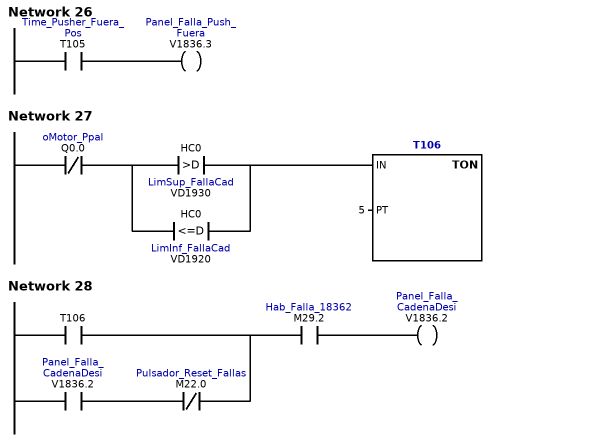
[picture p48: SBR20 networks 26-28]
Network 26
LD     Time_Pusher_Fuera_Pos:T105
=      Panel_Falla_Push_Fuera:V1836.3
Network 27
LDN    oMotor_Ppal:Q0.0
LDD>   HC0, LimSup_FallaCad:VD1930
OD<=   HC0, LimInf_FallaCad:VD1920
ALD
TON    T106, 5
Network 28
LD     T106
LD     Panel_Falla_CadenaDesi:V1836.2
AN     Pulsador_Reset_Fallas:M22.0
OLD
A      Hab_Falla_18362:M29.2
=      Panel_Falla_CadenaDesi:V1836.2
END_SUBROUTINE_BLOCK

SUBROUTINE_BLOCK Posiciones_Caja:SBR25
TITLE=
BEGIN
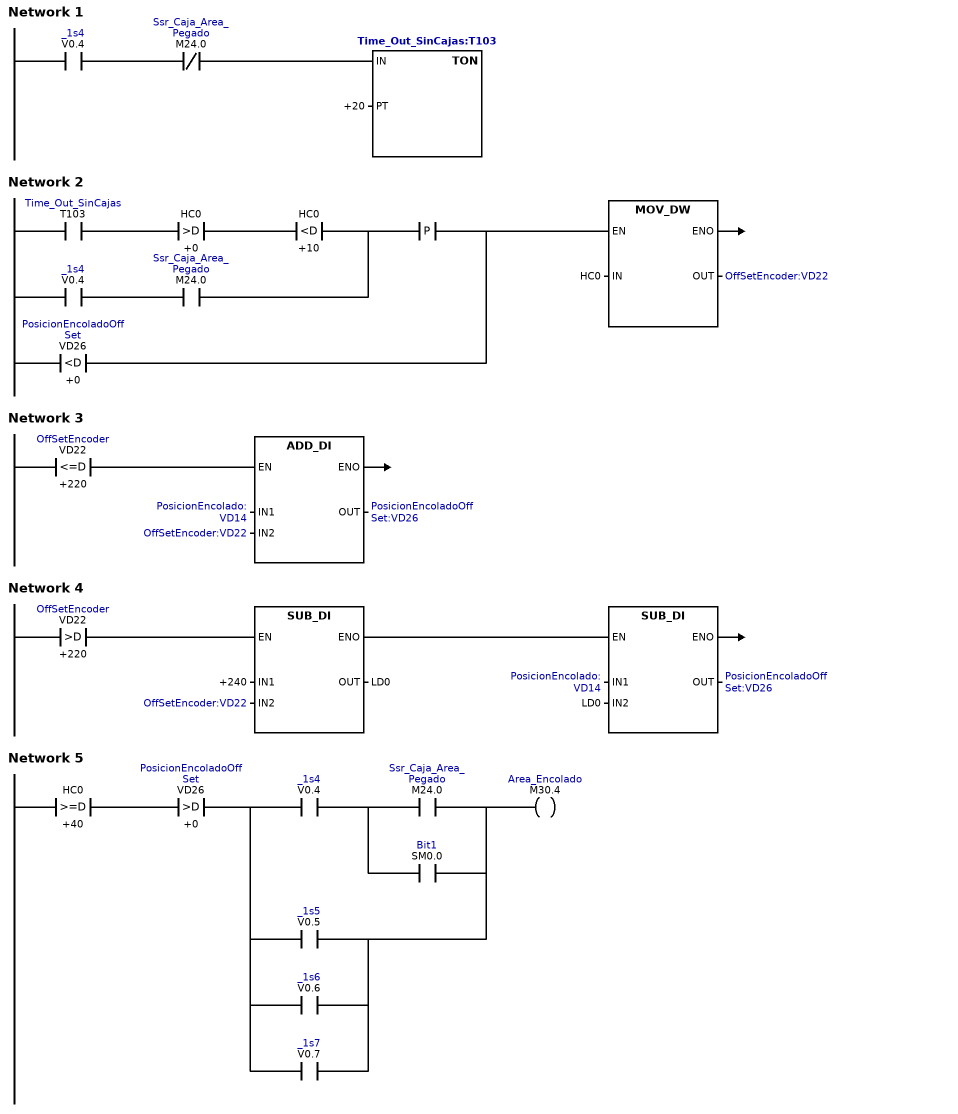
Network 1
LD     _1s4:V0.4
AN     Ssr_Caja_Area_Pegado:M24.0
TON    Time_Out_SinCajas:T103, +20
Network 2
LD     Time_Out_SinCajas:T103
AD>    HC0, +0
AD<    HC0, +10
LD     _1s4:V0.4
A      Ssr_Caja_Area_Pegado:M24.0
OLD
EU
OD<    PosicionEncoladoOffSet:VD26, +0
MOVD   HC0, OffSetEncoder:VD22
Network 3
LDD<=  OffSetEncoder:VD22, +220
MOVD   PosicionEncolado:VD14, PosicionEncoladoOffSet:VD26
+D     OffSetEncoder:VD22, PosicionEncoladoOffSet:VD26
Network 4
LDD>   OffSetEncoder:VD22, +220
MOVD   +240, LD0
AENO
-D     OffSetEncoder:VD22, LD0
AENO
MOVD   PosicionEncolado:VD14, PosicionEncoladoOffSet:VD26
-D     LD0, PosicionEncoladoOffSet:VD26
Network 5
LDD>=  HC0, +40
AD>    PosicionEncoladoOffSet:VD26, +0
LD     _1s4:V0.4
LD     Ssr_Caja_Area_Pegado:M24.0
O      Bit1:SM0.0
ALD
LD     _1s5:V0.5
O      _1s6:V0.6
O      _1s7:V0.7
OLD
ALD
=      Area_Encolado:M30.4
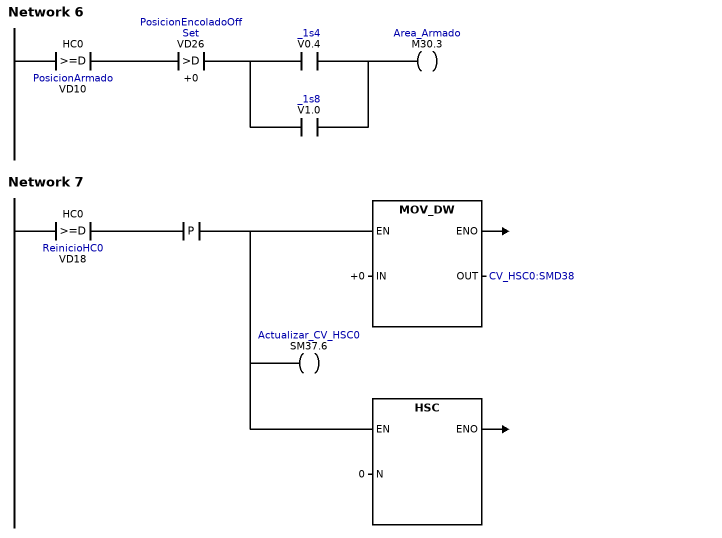
Network 6
LDD>=  HC0, PosicionArmado:VD10
AD>    PosicionEncoladoOffSet:VD26, +0
LD     _1s4:V0.4
O      _1s8:V1.0
ALD
=      Area_Armado:M30.3
Network 7
LDD>=  HC0, ReinicioHC0:VD18
EU
MOVD   +0, CV_HSC0:SMD38
=      Actualizar_CV_HSC0:SM37.6
HSC    0
END_SUBROUTINE_BLOCK

DATA_BLOCK_TAB USUARIO1
BEGIN
//COMENTARIOS DEL BLOQUE DE DATOS
//Pulse F1 para obtener Ayuda y un bloque de datos de ejemplo.
//****************************************************************
//****UTILIZO DE LAS WORDS DE 0 A 10 PARA LOS ESTADOS INTERNOS****
//****************************************************************
         _1sD1, 0            //Word de estados 1
         _2sw1, 0            //Word de estados 2
         _3sw1, 0            //Word de estados 3
         _4sw1, 0            //Word de estados 4
//****************************************************
//****UTILIZO DE LAS WORDS DE 10 A 100 PARA VARIOS****
//****************************************************
         PosicionArmado, 230 //Valor donde el encoder debe iniciar la secuencia de ARMADO
         PosicionEncolado, 5 //Valor donde el encoder debe iniciar la secuencia de PEGADO
         ReinicioHC0, 240    //Valor de reinicio del contador rapido HC0
         OffSetEncoder, 5    //Valor de Off set para cuentas encoder
         PosicionEncoladoOffSet, 0 //Valor para inicio Encolado con Off Set incluido
         WFallas, 0          //Word de FALLAS PARA PANEL!!!!
         Tiempo_Encolado_1, 9 //Tiempo x10ms de Encolado 1 en Uso
         Tiempo_Encolado_2, 7 //Tiempo x10ms de Encolado 2 en Uso
         Tiempo_NO_Encolar, 25 //Tiempo x10ms de NO ENCOLADO en Uso
//****************************************************
//Los tiempos en el panel tienen 2 decimales y el formato es entero
//por lo que el dato que envia el panel es multiplicado
//por 100 (ya que posee 2 decimales)
//y los timer tienen base de tiempo = 10ms por lo que no debo
//realizar ninguna cuenta auxiliar  
//En panel => 1,00 seg = 100 (dato al PLC)
//100 * 0.01 seg = 1 seg
//****************************************************
         Panel_Timer_Corte_Vacio, 5 //Tiempo de Corte de vacio desde panel
         Panel_Sel_Caja, 0   //Selección de Programa por Tipo de Caja
VW112    0                   //Libre
VW114    0                   //Libre
VW116    0                   //Libre
VW118    0                   //Libre
//**************************************************************************
// VD120  Utilizada para ver en el panel los valores actuales del encoder*** 
//**************************************************************************
VW124    0                   //Libre
VW126    0                   //Libre
VW128    0                   //Libre
//**********************************************************
//Estas words son para ajustar los tiempos
//mecanicos de la maquinas, aca figuran comentados
//pero en el programa se utilizan
//**********************************************************
         D_Pnel_T_Escuadre, 0 //Panel_TON_10 Timer Tiempo de Escuadre
         D_Pnel_T_RetardoPushe, 0 //Panel_TON_10 Timer Tiempo de Retardo de Pusher
         D_Pnel_T_Arranque_Bba, 10 //Panel_TON_100 Timer Tiempo Arranque Bomba Vacio
         D_Pnel_T_ArranqCyMPpal, 4 //Panel_TON_100 Timer Tiempo Arranque Cinta y Motor Ppal.
         D_Pnel_T_Falla_Pusher, 10 //Panel_TON_100 Timer Tiempo Falla Motor Pusher
         D_Pnel_T_FallaPistPush, 10 //Panel_TON_100 Timer Tiempo Falla Piston Pusher
//**********************************************************
// Valores de Encolado Ajustados desde Panel
// En este caso los datos llegan por 10ms como es la base del timer
//**********************************************************
         Panel_Tie_Enc_1_0, 9 //Tiempo x10ms de Encolado 1 Caja 15x1000
         Panel_Tie_Enc_2_0, 7 //Tiempo x10ms de Encolado 2 Caja 15x1000
         Panel_Tie_NoEnc_0, 25 //Tiempo x10ms de No Encolado Caja 15x1000
         Panel_Tie_Enc_1_1, 9 //Tiempo x10ms de Encolado 1 Caja 12x1500
         Panel_Tie_Enc_2_1, 7 //Tiempo x10ms de Encolado 2 Caja 12x1500
         Panel_Tie_NoEnc_1, 25 //Tiempo x10ms de No Encolado Caja 12x1500
         Panel_Tie_Enc_1_2, 9 //Tiempo x10ms de Encolado 1 Caja 12x1000
         Panel_Tie_Enc_2_2, 6 //Tiempo x10ms de Encolado 2 Caja 12x1000
         Panel_Tie_NoEnc_2, 18 //Tiempo x10ms de No Encolado Caja 12x1000
         Panel_Tie_Enc_1_3, 7 //Tiempo x10ms de Encolado 1 Caja 12x750
         Panel_Tie_Enc_2_3, 6 //Tiempo x10ms de Encolado 2 Caja 12x750
         Panel_Tie_NoEnc_3, 15 //Tiempo x10ms de No Encolado Caja 12x750
//*********************************************************************
// A PARTIR DE LA V1800 ARRANCO CON EL INTERCAMBIO DE DATOS CON EL PANEL 
// Ver simbolicos Standart Panel!!
//*********************************************************************
V1862    
V1862    
V1862    
V1862    
V1862    
V1862    
V1862    
V1862    
V1863    
V1863    
V1863    
V1863    
V1863    
V1863    
V1863    
V1863    
V1864    
V1864    
V1864    
V1864    
V1864    
V1864    
V1864    
V1864    
V1865    
V1865    
V1865    
V1865    
V1865    
V1865    
V1865    
V1865    
V1866    
V1866    
V1866    
V1866    
V1866    
V1866    
V1866    
V1866    
V1867    
V1867    
V1867    
V1867    
V1867    
V1867    
V1867    
V1867    
V1868    
V1868    
V1868    
V1868    
V1868    
V1868    
V1868    
V1868    
V1869    
V1869    
V1869    
V1869    
V1869    
V1869    
V1869    
V1869    
V1870    
V1870    
V1870    
V1870    
V1870    
V1870    
V1870    
V1870    
V1871    
V1871    
V1871    
V1871    
V1871    
V1871    
V1871    
V1871    
V1872    
V1872    
V1872    
V1872    
V1872    
V1872    
V1872    
V1872    
V1873    
V1873    
V1873    
V1873    
V1873    
V1873    
V1873    
V1873    
V1894    
V1894    
V1894    
V1894    
V1894    
V1894    
V1894    
V1894    
V1895    
V1895    
V1895    
V1895    
V1895    
V1895    
V1895    
V1895    
V1896    
V1896    
V1896    
V1896    
V1896    
V1896    
V1896    
V1896    
V1897    
V1897    
V1897    
V1897    
V1897    
V1897    
V1897    
V1897    
V1898    
V1898    
V1898    
V1898    
V1898    
V1898    
V1898    
V1898    
V1899    
V1899    
V1899    
V1899    
V1899    
V1899    
V1899    
V1899    
V1900    
V1900    
V1900    
V1900    
V1900    
V1900    
V1900    
V1900    
V1901    
V1901    
V1901    
V1901    
V1901    
V1901    
V1901    
V1901    
V1902    
V1902    
V1902    
V1902    
V1902    
V1902    
V1902    
V1902    
V1903    
V1903    
V1903    
V1903    
V1903    
V1903    
V1903    
V1903    
V1904    
V1904    
V1904    
V1904    
V1904    
V1904    
V1904    
V1904    
V1905    
V1905    
V1905    
V1905    
V1905    
V1905    
V1905    
V1905    
V1996    
V1996    
V1996    
V1996    
V1996    
V1996    
V1996    
V1996    
V1997    
V1997    
V1997    
V1997    
V1997    
V1997    
V1997    
V1997    
V1998    
V1998    
V1998    
V1998    
V1998    
V1998    
V1998    
V1998    
V1999    
V1999    
V1999    
V1999    
V1999    
V1999    
V1999    
V1999    
V2000    
V2000    
V2000    
V2000    
V2000    
V2000    
V2000    
V2000    
V2001    
V2001    
V2001    
V2001    
V2001    
V2001    
V2001    
V2001    
V2002    
V2002    
V2002    
V2002    
V2002    
V2002    
V2002    
V2002    
V2003    
V2003    
V2003    
V2003    
V2003    
V2003    
V2003    
V2003    
V2004    
V2004    
V2004    
V2004    
V2004    
V2004    
V2004    
V2004    
V2005    
V2005    
V2005    
V2005    
V2005    
V2005    
V2005    
V2005    
V2006    
V2006    
V2006    
V2006    
V2006    
V2006    
V2006    
V2006    
V2007    
V2007    
V2007    
V2007    
V2007    
V2007    
V2007    
V2007    
V2008    
V2008    
V2008    
V2008    
V2008    
V2008    
V2008    
V2008    
V2009    
V2009    
V2009    
V2009    
V2009    
V2009    
V2009    
V2009    
V2010    
V2010    
V2010    
V2010    
V2010    
V2010    
V2010    
V2010    
V2011    
V2011    
V2011    
V2011    
V2011    
V2011    
V2011    
V2011    
         dAux1
         ANUsrW00
         ANImgW02
         ANImgW04
         ANAvsW06
         ANAvsW08
         ANAvsW10
         ANAvsW12
         ANAvsW14
         ANAvsW16
         ANAvsW18
         ANAlaW20
         ANAlaW22
         ANAlaW24
         ANAlaW26
         ANAlaW28
         ANAlaW30
         ANAlaW32
         ANFalW34
         ANFalW36
         ANFalW38
         ANFalW40
         ANFalW42
         ANFalW44
         ANFalW46
         ANRecW48
         ANRecW50
         ANRecW52
         ANRecW54
         ANRecW56
         ANRecW58
         ANRecW60
         TcSisW00
         TcSisW02
         TcFunW00
         TcFunW02
         TcFunW04
         TcFunW06
         ImLedW00
         ImLedW02
         AxSisW00
         AxSisW02
         AxFunW00
         AxFunW02
         AxFunW04
         AxFunW06
         Res1890
         Res1892
         fTcSisW00
         fTcSisW02
         fTcFunW00
         fTcFunW02
         fTcFunW04
         fTcFunW06
         wLedRap
         wLedLen
         wLedPer
         wAux1
         wAux2
         wAux3
         wAux4
         wAux5
END_DATA_BLOCK_TAB
